# EPICS substitutions: iocs/AKD2GExample/iocBoot/iocAKD2GExample/asyn_motor.substitutions
file "$(MOTOR)/db/asyn_motor.db"
{
  pattern
  {M,  DTYP,        PORT,     ADDR,  DESC,    EGU,      DIR,  VMAX,  VELO,  VBAS,  ACCL,  BDST,     BVEL,  BACC,     MRES,      PREC,  DHLM,       DLLM,   INIT}
  { m1, "asynMotor", AKD2G1,   0,    "Motor 1",    um,       Pos,  15.,   3.,    .05,    .5,    0,       1.0,    2,    .001,    9,   0,       0,  ""}
}
